PROGRAM MedidaDiamMec
VAR
	LoopCounter:INT;
	
	//Variables para la lectura de sensores
	MedSenMec:REAL:=0.0;
	MS1:REAL:=0.0;
	MS2:REAL:=0.0;
	
	//Variables para la media de medidas de los sensores
	Lecturas:ARRAY[0..9] OF REAL:=[10(0.0)]; 	//Medidas del diametro inicializadas
	Index:INT:=0; 								//Indice del vector de medidas 
	Suma:REAL:=0.0; 							//Suma de medidas
	
END_VAR

//Calculo del diametro
MS1:=-0.02157*IO.I_SMec1+5.82;	//Paso de medida leida por tarjeta a mm
MS2:=-0.02157*IO.I_SMec2+5.82;	//Paso de medida leida por tarjeta a mm
MedSenMec:=((MS1+MS2)/2);

//Hacer media de las 10 ultimas medidas del diametro
Suma:= Suma - Lecturas[Index];
Lecturas[index]:=MedSenMec;
Suma:=Suma+Lecturas[index];
Index:= Index + 1;
IF (Index > 9) THEN
	Index := 0;    	//Volvemos al inicio del vector
END_IF
GVL.MedidaSensorMecanico:=Suma/10;

END_PROGRAM

(* stored: Version 1.1.0.1, ProductVersion 3.1.4024.9
   POU MedidaDiamMec: Id {e0677ec7-582d-4897-a836-e9af0d4a41cf}, SpecialFunc None *)
